FUNCTION TryConvert_LINT_TO_TIME : BOOL
VAR_INPUT
	in : LINT;
	out : REFERENCE TO TIME;
END_VAR

IF in > DatatypeLimits.MAX_VALUE_OF_LINT_WHICH_CAN_BE_HELD_IN_A_TIME THEN
	RETURN;
END_IF

IF in < DatatypeLimits.MIN_VALUE_OF_LINT_WHICH_CAN_BE_HELD_IN_A_TIME THEN
	RETURN;
END_IF

out := LINT_TO_TIME(in);
TryConvert_LINT_TO_TIME := TRUE;

END_FUNCTION

(* stored: Version 1.1.0.1, ProductVersion 3.1.4024.12
   POU TryConvert_LINT_TO_TIME: Id {f760f609-ea98-449f-8fd9-217fede4fb66}, SpecialFunc None *)
